TYPE U_UMC_Lenze_Status :
UNION
	Input		: UINT;	
	Data		: T_UMC_Lenze_Status;
END_UNION
END_TYPE

(* stored: Version 1.1.0.1, ProductVersion 3.1.0.19
   DUT U_UMC_Lenze_Status: Id {a9ec2edf-c91d-463f-b398-3e68d1d88a6f} *)
